PROGRAM WriteAnalogOutput
VAR
	temp: REAL;
END_VAR

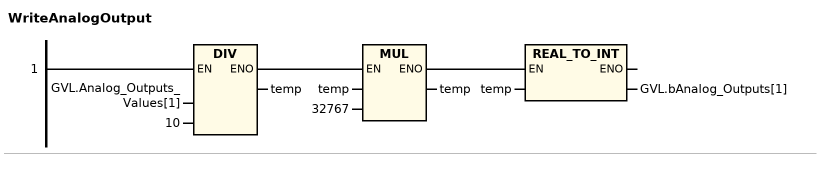
// NETWORK 1
temp := GVL.Analog_Outputs_Values[1] / 10;
temp := temp * 32767;
GVL.bAnalog_Outputs[1] := REAL_TO_INT(temp);

END_PROGRAM

(* stored: Version 1.1.0.1, ProductVersion 3.1.4024.12
   POU WriteAnalogOutput: Id {a9a89dd7-60b8-48eb-aa66-96c576096e6c}, SpecialFunc None *)
